// TIA Portal V21 export
TYPE "Std_Conteggi"
   STRUCT
      Dati : Struct
         MemStatoIngConteggio : Bool;
         ActConteggio : DInt;
         SimulazioneIngresso : Bool;
      END_STRUCT;
   END_STRUCT;
END_TYPE
